Staubli VAL3: clearScreen.pgx

public program clearScreen()
begin

  // Do nothing
  // See start() program for more details

end
